# EPICS StreamDevice protocol: src/main/epics/protocol/Lidar.proto
# PuddlePeeker.proto
Terminator = LF;
ReadTimeout = 200;

get_temperature {
   out "T?";
   in "T %f";
   ExtraInput=Ignore;
}
get_distance {
   out "D?";
   in "D %f %(\$1)f";
   ExtraInput=Ignore;
}
